TYPE raPositions :
STRUCT
	cor: INT;
	color: DWORD;
END_STRUCT
END_TYPE

(* stored: Version 1.1.0.1, ProductVersion 3.1.4024.12
   DUT raPositions: Id {88a9e68e-bdfa-42f0-b7df-f54994d483a5} *)
